function_block FB_Syntax_Derived extends FB_Syntax_AbstractBase implements I_Syntax_Extended
var
    _sStatus : string := 'IDLE';
    _nCounter : dint;
end_var

_nCounter := _nCounter + 1;

method M_Execute : bool
var_input
    nCommand : dint;
end_var
case nCommand of
    1:
        _sStatus := 'RUNNING';
    2:
        _sStatus := 'PAUSED';
else
    _sStatus := 'UNKNOWN';
end_case
M_Execute := true;
END_METHOD

method M_GetValue : int
M_GetValue := TO_INT(_nCounter);
END_METHOD

method M_Reset : bool
_nCounter := 0;
_bReady := TRUE;
_sStatus := 'RESET';
M_Reset := TRUE;
END_METHOD

property P_ExtendedStatus : int
GET
var
end_var
P_ExtendedStatus := 1;
END_GET
END_PROPERTY

property P_Status : string
GET
var
end_var
P_Status := _sStatus;
END_GET
END_PROPERTY

END_FUNCTION_BLOCK

(* stored: Version 1.1.0.1, ProductVersion 3.1.4024.16
   POU FB_Syntax_Derived: Id {ee893be3-3f4d-43fd-ad98-be9638564c28}, SpecialFunc None
   Method M_Execute: Id {e5f6a1b2-c3d4-4e5f-c06b-7c8d9e0f1a2b}
   Method M_GetValue: Id {ab1b6ad1-a4ee-40bd-81ae-4c3f57901aec}
   Method M_Reset: Id {d4e5f6a1-b2c3-4d4e-bf5a-6b7c8d9e0f1a}
   Property P_ExtendedStatus: Id {acb160f8-190f-4161-806f-16a237f4e6af}
   Get Get: Id {5e573bf0-7431-42eb-99fa-2e7219b3fa95}
   Property P_Status: Id {f6a1b2c3-d4e5-4f6a-d17c-8d9e0f1a2b3c}
   Get Get: Id {a1b2c3d4-e5f6-4a7b-e28d-9e0f1a2b3c4d} *)
